TYPE TcoKeyMode_Status :
STRUCT
	ActionDescription : STRING(100);	

END_STRUCT
END_TYPE

(* stored: Version 1.1.0.1
   DUT TcoKeyMode_Status: Id {5e0c957e-ef4f-47ec-b418-83717285b373} *)
